// TIA Portal V16 export
// export: Created 2021-11-12T13:31:08.2127898Z, ExportSetting WithDefaults, DisplayName Totally Integrated Automation Portal, DisplayVersion V16 Update 3, DisplayName TIA Portal Version Control Interface, DisplayVersion V16 Update 2, DisplayName TIA Portal Openness, DisplayVersion V16 Update 3, DisplayName SINAMICS Startdrive Advanced, DisplayVersion V16 Update 5, DisplayName SINAMICS Startdrive G130, G150, S120, S150, SINAMICS MV, S210, DisplayVersion V16 Update 5, DisplayName SINAMICS Startdrive G110M, G120, G120C, G120D, G120P, G115D, DisplayVersion V16 Update 5, DisplayName STEP 7 Professional, DisplayVersion V16 Update 3, DisplayName STEP 7 Safety, DisplayVersion V16, DisplayName WinCC UA Professional, DisplayVersion V16 Update 3
FUNCTION_BLOCK "Main_Safety_RTG1"   // FB1, F_LAD
{ S7_Optimized_Access := 'TRUE' }
VERSION : 0.1
// stored: AutoNumber false, IsIECCheckEnabled false, UDAEnableTagReadback false
BEGIN

REGION Network 1: *************** Ingoing communication section start ***************
END_REGION

REGION Network 2: Communication: BSN1 / BSN2 -> CRS
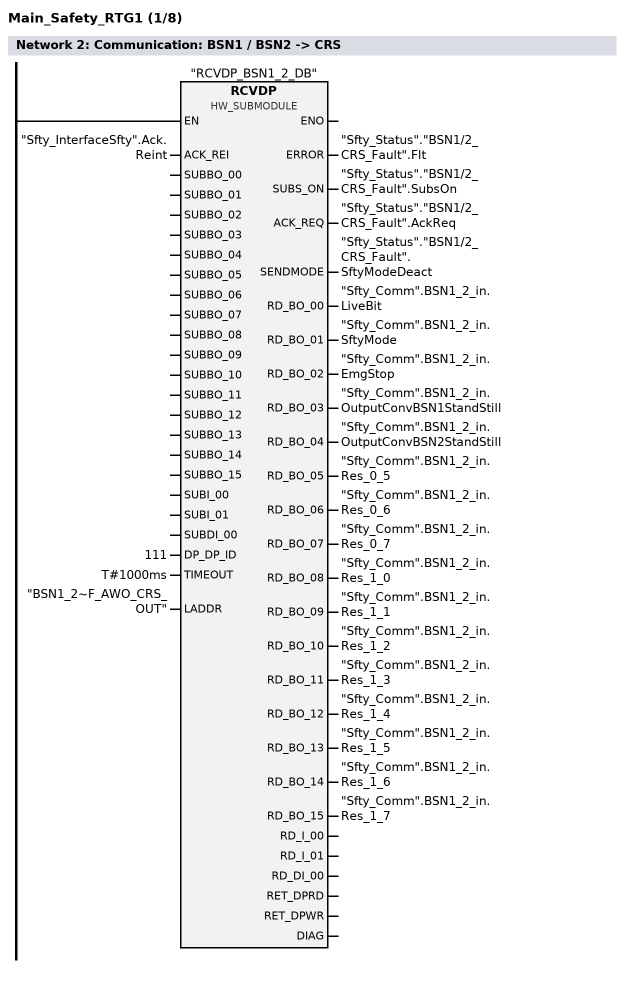
   RUNG wire#powerrail
      { S7_Templates := "laddr_type := HW_SUBMODULE" } "RCVDP_BSN1_2_DB".RCVDP(ACK_REI := "Sfty_InterfaceSfty".Ack.Reint, SUBBO_00 :=, SUBBO_01 :=, SUBBO_02 :=, SUBBO_03 :=, SUBBO_04 :=, SUBBO_05 :=, SUBBO_06 :=, SUBBO_07 :=, SUBBO_08 :=, SUBBO_09 :=, SUBBO_10 :=, SUBBO_11 :=, SUBBO_12 :=, SUBBO_13 :=, SUBBO_14 :=, SUBBO_15 :=, SUBI_00 :=, SUBI_01 :=, SUBDI_00 :=, DP_DP_ID := 111, TIMEOUT := T#1000ms, LADDR := "BSN1_2~F_AWO_CRS_OUT", ERROR => "Sfty_Status"."BSN1/2_CRS_Fault".Flt, SUBS_ON => "Sfty_Status"."BSN1/2_CRS_Fault".SubsOn, ACK_REQ => "Sfty_Status"."BSN1/2_CRS_Fault".AckReq, SENDMODE => "Sfty_Status"."BSN1/2_CRS_Fault".SftyModeDeact, RD_BO_00 => "Sfty_Comm".BSN1_2_in.LiveBit, RD_BO_01 => "Sfty_Comm".BSN1_2_in.SftyMode, RD_BO_02 => "Sfty_Comm".BSN1_2_in.EmgStop, RD_BO_03 => "Sfty_Comm".BSN1_2_in.OutputConvBSN1StandStill, RD_BO_04 => "Sfty_Comm".BSN1_2_in.OutputConvBSN2StandStill, RD_BO_05 => "Sfty_Comm".BSN1_2_in.Res_0_5, RD_BO_06 => "Sfty_Comm".BSN1_2_in.Res_0_6, RD_BO_07 => "Sfty_Comm".BSN1_2_in.Res_0_7, RD_BO_08 => "Sfty_Comm".BSN1_2_in.Res_1_0, RD_BO_09 => "Sfty_Comm".BSN1_2_in.Res_1_1, RD_BO_10 => "Sfty_Comm".BSN1_2_in.Res_1_2, RD_BO_11 => "Sfty_Comm".BSN1_2_in.Res_1_3, RD_BO_12 => "Sfty_Comm".BSN1_2_in.Res_1_4, RD_BO_13 => "Sfty_Comm".BSN1_2_in.Res_1_5, RD_BO_14 => "Sfty_Comm".BSN1_2_in.Res_1_6, RD_BO_15 => "Sfty_Comm".BSN1_2_in.Res_1_7, RD_I_00 =>, RD_I_01 =>, RD_DI_00 =>, RET_DPRD =>, RET_DPWR =>, DIAG =>)
   END_RUNG
   // the same network as SCL:
   "RCVDP_BSN1_2_DB"(ACK_REI := "Sfty_InterfaceSfty".Ack.Reint,   // RCVDP
                     DP_DP_ID := 111,
                     TIMEOUT := T#1000ms,
                     LADDR := "BSN1_2~F_AWO_CRS_OUT",
                     ERROR => "Sfty_Status"."BSN1/2_CRS_Fault".Flt,
                     SUBS_ON => "Sfty_Status"."BSN1/2_CRS_Fault".SubsOn,
                     ACK_REQ => "Sfty_Status"."BSN1/2_CRS_Fault".AckReq,
                     SENDMODE => "Sfty_Status"."BSN1/2_CRS_Fault".SftyModeDeact,
                     RD_BO_00 => "Sfty_Comm".BSN1_2_in.LiveBit,
                     RD_BO_01 => "Sfty_Comm".BSN1_2_in.SftyMode,
                     RD_BO_02 => "Sfty_Comm".BSN1_2_in.EmgStop,
                     RD_BO_03 => "Sfty_Comm".BSN1_2_in.OutputConvBSN1StandStill,
                     RD_BO_04 => "Sfty_Comm".BSN1_2_in.OutputConvBSN2StandStill,
                     RD_BO_05 => "Sfty_Comm".BSN1_2_in.Res_0_5,
                     RD_BO_06 => "Sfty_Comm".BSN1_2_in.Res_0_6,
                     RD_BO_07 => "Sfty_Comm".BSN1_2_in.Res_0_7,
                     RD_BO_08 => "Sfty_Comm".BSN1_2_in.Res_1_0,
                     RD_BO_09 => "Sfty_Comm".BSN1_2_in.Res_1_1,
                     RD_BO_10 => "Sfty_Comm".BSN1_2_in.Res_1_2,
                     RD_BO_11 => "Sfty_Comm".BSN1_2_in.Res_1_3,
                     RD_BO_12 => "Sfty_Comm".BSN1_2_in.Res_1_4,
                     RD_BO_13 => "Sfty_Comm".BSN1_2_in.Res_1_5,
                     RD_BO_14 => "Sfty_Comm".BSN1_2_in.Res_1_6,
                     RD_BO_15 => "Sfty_Comm".BSN1_2_in.Res_1_7);
END_REGION

REGION Network 3: Communication: SCH1 -> CRS
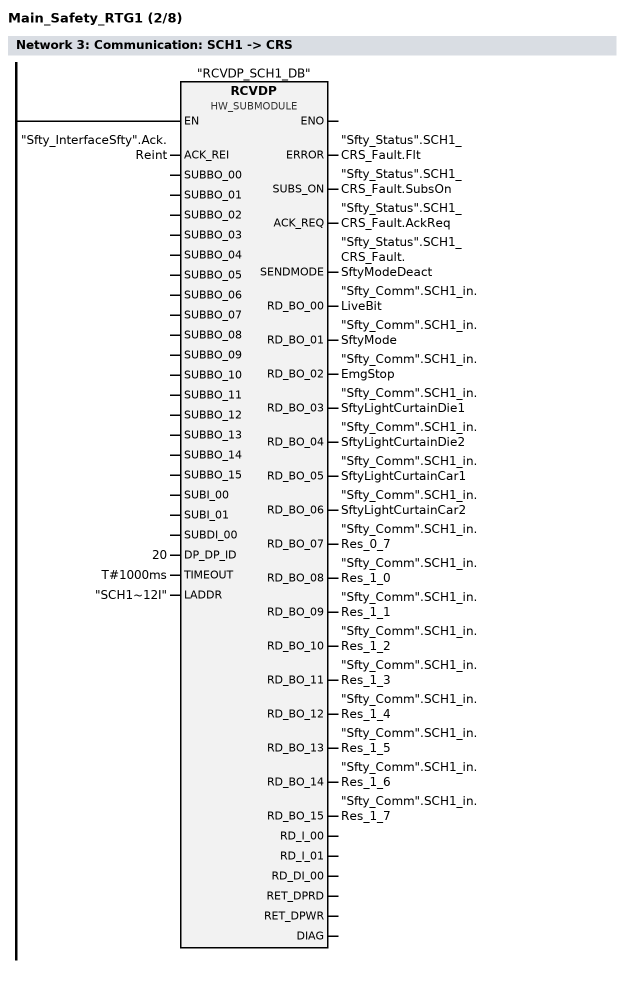
   RUNG wire#powerrail
      { S7_Templates := "laddr_type := HW_SUBMODULE" } "RCVDP_SCH1_DB".RCVDP(ACK_REI := "Sfty_InterfaceSfty".Ack.Reint, SUBBO_00 :=, SUBBO_01 :=, SUBBO_02 :=, SUBBO_03 :=, SUBBO_04 :=, SUBBO_05 :=, SUBBO_06 :=, SUBBO_07 :=, SUBBO_08 :=, SUBBO_09 :=, SUBBO_10 :=, SUBBO_11 :=, SUBBO_12 :=, SUBBO_13 :=, SUBBO_14 :=, SUBBO_15 :=, SUBI_00 :=, SUBI_01 :=, SUBDI_00 :=, DP_DP_ID := 20, TIMEOUT := T#1000ms, LADDR := "SCH1~12I", ERROR => "Sfty_Status".SCH1_CRS_Fault.Flt, SUBS_ON => "Sfty_Status".SCH1_CRS_Fault.SubsOn, ACK_REQ => "Sfty_Status".SCH1_CRS_Fault.AckReq, SENDMODE => "Sfty_Status".SCH1_CRS_Fault.SftyModeDeact, RD_BO_00 => "Sfty_Comm".SCH1_in.LiveBit, RD_BO_01 => "Sfty_Comm".SCH1_in.SftyMode, RD_BO_02 => "Sfty_Comm".SCH1_in.EmgStop, RD_BO_03 => "Sfty_Comm".SCH1_in.SftyLightCurtainDie1, RD_BO_04 => "Sfty_Comm".SCH1_in.SftyLightCurtainDie2, RD_BO_05 => "Sfty_Comm".SCH1_in.SftyLightCurtainCar1, RD_BO_06 => "Sfty_Comm".SCH1_in.SftyLightCurtainCar2, RD_BO_07 => "Sfty_Comm".SCH1_in.Res_0_7, RD_BO_08 => "Sfty_Comm".SCH1_in.Res_1_0, RD_BO_09 => "Sfty_Comm".SCH1_in.Res_1_1, RD_BO_10 => "Sfty_Comm".SCH1_in.Res_1_2, RD_BO_11 => "Sfty_Comm".SCH1_in.Res_1_3, RD_BO_12 => "Sfty_Comm".SCH1_in.Res_1_4, RD_BO_13 => "Sfty_Comm".SCH1_in.Res_1_5, RD_BO_14 => "Sfty_Comm".SCH1_in.Res_1_6, RD_BO_15 => "Sfty_Comm".SCH1_in.Res_1_7, RD_I_00 =>, RD_I_01 =>, RD_DI_00 =>, RET_DPRD =>, RET_DPWR =>, DIAG =>)
   END_RUNG
   // the same network as SCL:
   "RCVDP_SCH1_DB"(ACK_REI := "Sfty_InterfaceSfty".Ack.Reint,   // RCVDP
                   DP_DP_ID := 20,
                   TIMEOUT := T#1000ms,
                   LADDR := "SCH1~12I",
                   ERROR => "Sfty_Status".SCH1_CRS_Fault.Flt,
                   SUBS_ON => "Sfty_Status".SCH1_CRS_Fault.SubsOn,
                   ACK_REQ => "Sfty_Status".SCH1_CRS_Fault.AckReq,
                   SENDMODE => "Sfty_Status".SCH1_CRS_Fault.SftyModeDeact,
                   RD_BO_00 => "Sfty_Comm".SCH1_in.LiveBit,
                   RD_BO_01 => "Sfty_Comm".SCH1_in.SftyMode,
                   RD_BO_02 => "Sfty_Comm".SCH1_in.EmgStop,
                   RD_BO_03 => "Sfty_Comm".SCH1_in.SftyLightCurtainDie1,
                   RD_BO_04 => "Sfty_Comm".SCH1_in.SftyLightCurtainDie2,
                   RD_BO_05 => "Sfty_Comm".SCH1_in.SftyLightCurtainCar1,
                   RD_BO_06 => "Sfty_Comm".SCH1_in.SftyLightCurtainCar2,
                   RD_BO_07 => "Sfty_Comm".SCH1_in.Res_0_7,
                   RD_BO_08 => "Sfty_Comm".SCH1_in.Res_1_0,
                   RD_BO_09 => "Sfty_Comm".SCH1_in.Res_1_1,
                   RD_BO_10 => "Sfty_Comm".SCH1_in.Res_1_2,
                   RD_BO_11 => "Sfty_Comm".SCH1_in.Res_1_3,
                   RD_BO_12 => "Sfty_Comm".SCH1_in.Res_1_4,
                   RD_BO_13 => "Sfty_Comm".SCH1_in.Res_1_5,
                   RD_BO_14 => "Sfty_Comm".SCH1_in.Res_1_6,
                   RD_BO_15 => "Sfty_Comm".SCH1_in.Res_1_7);
END_REGION

REGION Network 4: Communication: BSN3 -> CRS
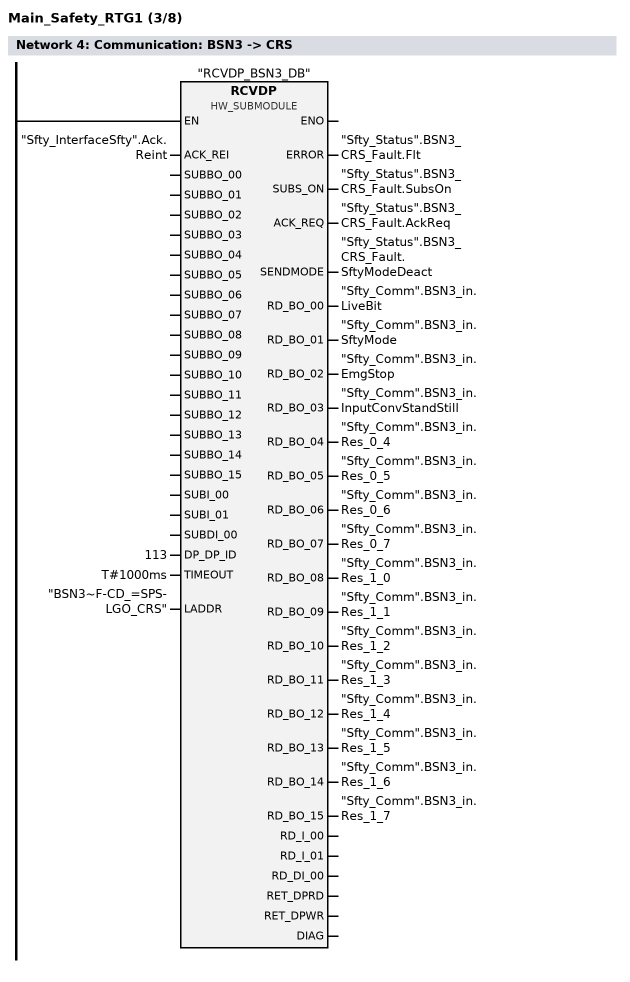
   RUNG wire#powerrail
      { S7_Templates := "laddr_type := HW_SUBMODULE" } "RCVDP_BSN3_DB".RCVDP(ACK_REI := "Sfty_InterfaceSfty".Ack.Reint, SUBBO_00 :=, SUBBO_01 :=, SUBBO_02 :=, SUBBO_03 :=, SUBBO_04 :=, SUBBO_05 :=, SUBBO_06 :=, SUBBO_07 :=, SUBBO_08 :=, SUBBO_09 :=, SUBBO_10 :=, SUBBO_11 :=, SUBBO_12 :=, SUBBO_13 :=, SUBBO_14 :=, SUBBO_15 :=, SUBI_00 :=, SUBI_01 :=, SUBDI_00 :=, DP_DP_ID := 113, TIMEOUT := T#1000ms, LADDR := "BSN3~F-CD_=SPS-LGO_CRS", ERROR => "Sfty_Status".BSN3_CRS_Fault.Flt, SUBS_ON => "Sfty_Status".BSN3_CRS_Fault.SubsOn, ACK_REQ => "Sfty_Status".BSN3_CRS_Fault.AckReq, SENDMODE => "Sfty_Status".BSN3_CRS_Fault.SftyModeDeact, RD_BO_00 => "Sfty_Comm".BSN3_in.LiveBit, RD_BO_01 => "Sfty_Comm".BSN3_in.SftyMode, RD_BO_02 => "Sfty_Comm".BSN3_in.EmgStop, RD_BO_03 => "Sfty_Comm".BSN3_in.InputConvStandStill, RD_BO_04 => "Sfty_Comm".BSN3_in.Res_0_4, RD_BO_05 => "Sfty_Comm".BSN3_in.Res_0_5, RD_BO_06 => "Sfty_Comm".BSN3_in.Res_0_6, RD_BO_07 => "Sfty_Comm".BSN3_in.Res_0_7, RD_BO_08 => "Sfty_Comm".BSN3_in.Res_1_0, RD_BO_09 => "Sfty_Comm".BSN3_in.Res_1_1, RD_BO_10 => "Sfty_Comm".BSN3_in.Res_1_2, RD_BO_11 => "Sfty_Comm".BSN3_in.Res_1_3, RD_BO_12 => "Sfty_Comm".BSN3_in.Res_1_4, RD_BO_13 => "Sfty_Comm".BSN3_in.Res_1_5, RD_BO_14 => "Sfty_Comm".BSN3_in.Res_1_6, RD_BO_15 => "Sfty_Comm".BSN3_in.Res_1_7, RD_I_00 =>, RD_I_01 =>, RD_DI_00 =>, RET_DPRD =>, RET_DPWR =>, DIAG =>)
   END_RUNG
   // the same network as SCL:
   "RCVDP_BSN3_DB"(ACK_REI := "Sfty_InterfaceSfty".Ack.Reint,   // RCVDP
                   DP_DP_ID := 113,
                   TIMEOUT := T#1000ms,
                   LADDR := "BSN3~F-CD_=SPS-LGO_CRS",
                   ERROR => "Sfty_Status".BSN3_CRS_Fault.Flt,
                   SUBS_ON => "Sfty_Status".BSN3_CRS_Fault.SubsOn,
                   ACK_REQ => "Sfty_Status".BSN3_CRS_Fault.AckReq,
                   SENDMODE => "Sfty_Status".BSN3_CRS_Fault.SftyModeDeact,
                   RD_BO_00 => "Sfty_Comm".BSN3_in.LiveBit,
                   RD_BO_01 => "Sfty_Comm".BSN3_in.SftyMode,
                   RD_BO_02 => "Sfty_Comm".BSN3_in.EmgStop,
                   RD_BO_03 => "Sfty_Comm".BSN3_in.InputConvStandStill,
                   RD_BO_04 => "Sfty_Comm".BSN3_in.Res_0_4,
                   RD_BO_05 => "Sfty_Comm".BSN3_in.Res_0_5,
                   RD_BO_06 => "Sfty_Comm".BSN3_in.Res_0_6,
                   RD_BO_07 => "Sfty_Comm".BSN3_in.Res_0_7,
                   RD_BO_08 => "Sfty_Comm".BSN3_in.Res_1_0,
                   RD_BO_09 => "Sfty_Comm".BSN3_in.Res_1_1,
                   RD_BO_10 => "Sfty_Comm".BSN3_in.Res_1_2,
                   RD_BO_11 => "Sfty_Comm".BSN3_in.Res_1_3,
                   RD_BO_12 => "Sfty_Comm".BSN3_in.Res_1_4,
                   RD_BO_13 => "Sfty_Comm".BSN3_in.Res_1_5,
                   RD_BO_14 => "Sfty_Comm".BSN3_in.Res_1_6,
                   RD_BO_15 => "Sfty_Comm".BSN3_in.Res_1_7);
END_REGION

REGION Network 5: Communication: BSN4 / BSN5 -> CRS
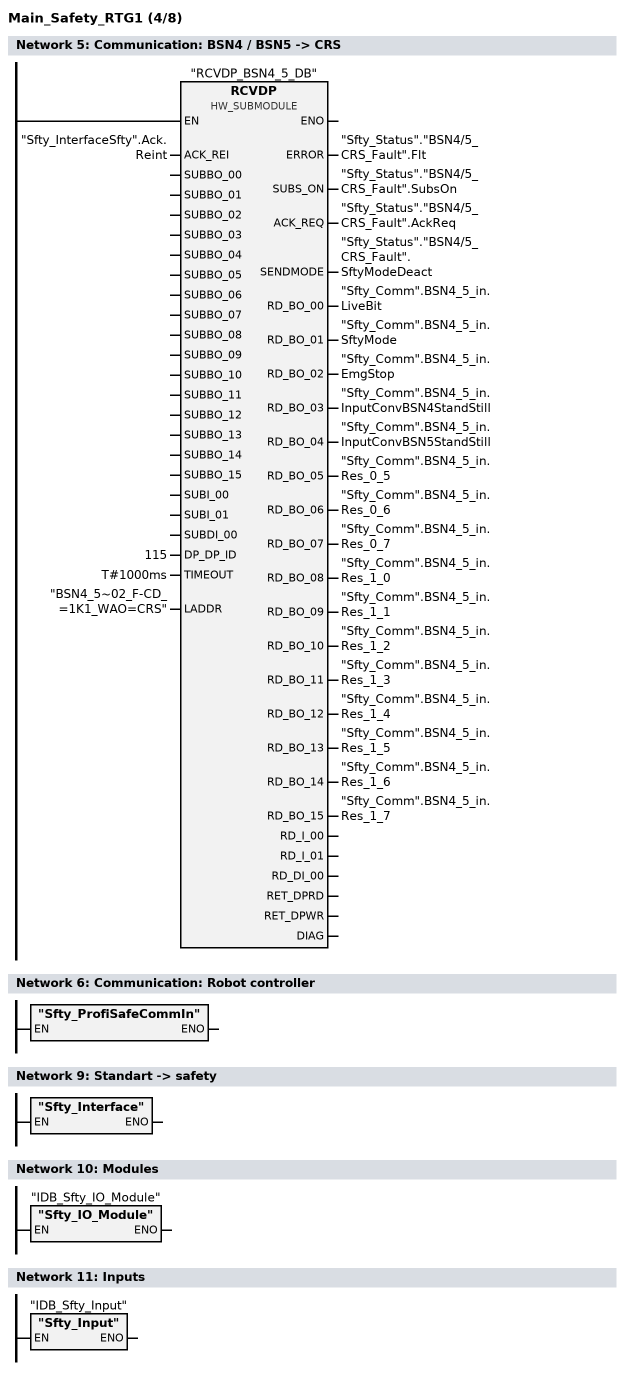
   RUNG wire#powerrail
      { S7_Templates := "laddr_type := HW_SUBMODULE" } "RCVDP_BSN4_5_DB".RCVDP(ACK_REI := "Sfty_InterfaceSfty".Ack.Reint, SUBBO_00 :=, SUBBO_01 :=, SUBBO_02 :=, SUBBO_03 :=, SUBBO_04 :=, SUBBO_05 :=, SUBBO_06 :=, SUBBO_07 :=, SUBBO_08 :=, SUBBO_09 :=, SUBBO_10 :=, SUBBO_11 :=, SUBBO_12 :=, SUBBO_13 :=, SUBBO_14 :=, SUBBO_15 :=, SUBI_00 :=, SUBI_01 :=, SUBDI_00 :=, DP_DP_ID := 115, TIMEOUT := T#1000ms, LADDR := "BSN4_5~02_F-CD_=1K1_WAO=CRS", ERROR => "Sfty_Status"."BSN4/5_CRS_Fault".Flt, SUBS_ON => "Sfty_Status"."BSN4/5_CRS_Fault".SubsOn, ACK_REQ => "Sfty_Status"."BSN4/5_CRS_Fault".AckReq, SENDMODE => "Sfty_Status"."BSN4/5_CRS_Fault".SftyModeDeact, RD_BO_00 => "Sfty_Comm".BSN4_5_in.LiveBit, RD_BO_01 => "Sfty_Comm".BSN4_5_in.SftyMode, RD_BO_02 => "Sfty_Comm".BSN4_5_in.EmgStop, RD_BO_03 => "Sfty_Comm".BSN4_5_in.InputConvBSN4StandStill, RD_BO_04 => "Sfty_Comm".BSN4_5_in.InputConvBSN5StandStill, RD_BO_05 => "Sfty_Comm".BSN4_5_in.Res_0_5, RD_BO_06 => "Sfty_Comm".BSN4_5_in.Res_0_6, RD_BO_07 => "Sfty_Comm".BSN4_5_in.Res_0_7, RD_BO_08 => "Sfty_Comm".BSN4_5_in.Res_1_0, RD_BO_09 => "Sfty_Comm".BSN4_5_in.Res_1_1, RD_BO_10 => "Sfty_Comm".BSN4_5_in.Res_1_2, RD_BO_11 => "Sfty_Comm".BSN4_5_in.Res_1_3, RD_BO_12 => "Sfty_Comm".BSN4_5_in.Res_1_4, RD_BO_13 => "Sfty_Comm".BSN4_5_in.Res_1_5, RD_BO_14 => "Sfty_Comm".BSN4_5_in.Res_1_6, RD_BO_15 => "Sfty_Comm".BSN4_5_in.Res_1_7, RD_I_00 =>, RD_I_01 =>, RD_DI_00 =>, RET_DPRD =>, RET_DPWR =>, DIAG =>)
   END_RUNG
   // the same network as SCL:
   "RCVDP_BSN4_5_DB"(ACK_REI := "Sfty_InterfaceSfty".Ack.Reint,   // RCVDP
                     DP_DP_ID := 115,
                     TIMEOUT := T#1000ms,
                     LADDR := "BSN4_5~02_F-CD_=1K1_WAO=CRS",
                     ERROR => "Sfty_Status"."BSN4/5_CRS_Fault".Flt,
                     SUBS_ON => "Sfty_Status"."BSN4/5_CRS_Fault".SubsOn,
                     ACK_REQ => "Sfty_Status"."BSN4/5_CRS_Fault".AckReq,
                     SENDMODE => "Sfty_Status"."BSN4/5_CRS_Fault".SftyModeDeact,
                     RD_BO_00 => "Sfty_Comm".BSN4_5_in.LiveBit,
                     RD_BO_01 => "Sfty_Comm".BSN4_5_in.SftyMode,
                     RD_BO_02 => "Sfty_Comm".BSN4_5_in.EmgStop,
                     RD_BO_03 => "Sfty_Comm".BSN4_5_in.InputConvBSN4StandStill,
                     RD_BO_04 => "Sfty_Comm".BSN4_5_in.InputConvBSN5StandStill,
                     RD_BO_05 => "Sfty_Comm".BSN4_5_in.Res_0_5,
                     RD_BO_06 => "Sfty_Comm".BSN4_5_in.Res_0_6,
                     RD_BO_07 => "Sfty_Comm".BSN4_5_in.Res_0_7,
                     RD_BO_08 => "Sfty_Comm".BSN4_5_in.Res_1_0,
                     RD_BO_09 => "Sfty_Comm".BSN4_5_in.Res_1_1,
                     RD_BO_10 => "Sfty_Comm".BSN4_5_in.Res_1_2,
                     RD_BO_11 => "Sfty_Comm".BSN4_5_in.Res_1_3,
                     RD_BO_12 => "Sfty_Comm".BSN4_5_in.Res_1_4,
                     RD_BO_13 => "Sfty_Comm".BSN4_5_in.Res_1_5,
                     RD_BO_14 => "Sfty_Comm".BSN4_5_in.Res_1_6,
                     RD_BO_15 => "Sfty_Comm".BSN4_5_in.Res_1_7);
END_REGION

REGION Network 6: Communication: Robot controller
   RUNG wire#powerrail
      "Sfty_ProfiSafeCommIn"()
   END_RUNG
   // the same network as SCL:
   "Sfty_ProfiSafeCommIn"();
END_REGION

REGION Network 7: *************** Ingoing communication section end ***************
END_REGION

REGION Network 8: *************** Interface ***************
END_REGION

REGION Network 9: Standart -> safety
   RUNG wire#powerrail
      "Sfty_Interface"()
   END_RUNG
   // the same network as SCL:
   "Sfty_Interface"();
END_REGION

REGION Network 10: Modules
   RUNG wire#powerrail
      "IDB_Sfty_IO_Module"()
   END_RUNG
   // the same network as SCL:
   "IDB_Sfty_IO_Module"();   // "Sfty_IO_Module"
END_REGION

REGION Network 11: Inputs
   RUNG wire#powerrail
      "IDB_Sfty_Input"()
   END_RUNG
   // the same network as SCL:
   "IDB_Sfty_Input"();   // "Sfty_Input"
END_REGION

REGION Network 12: Outputs
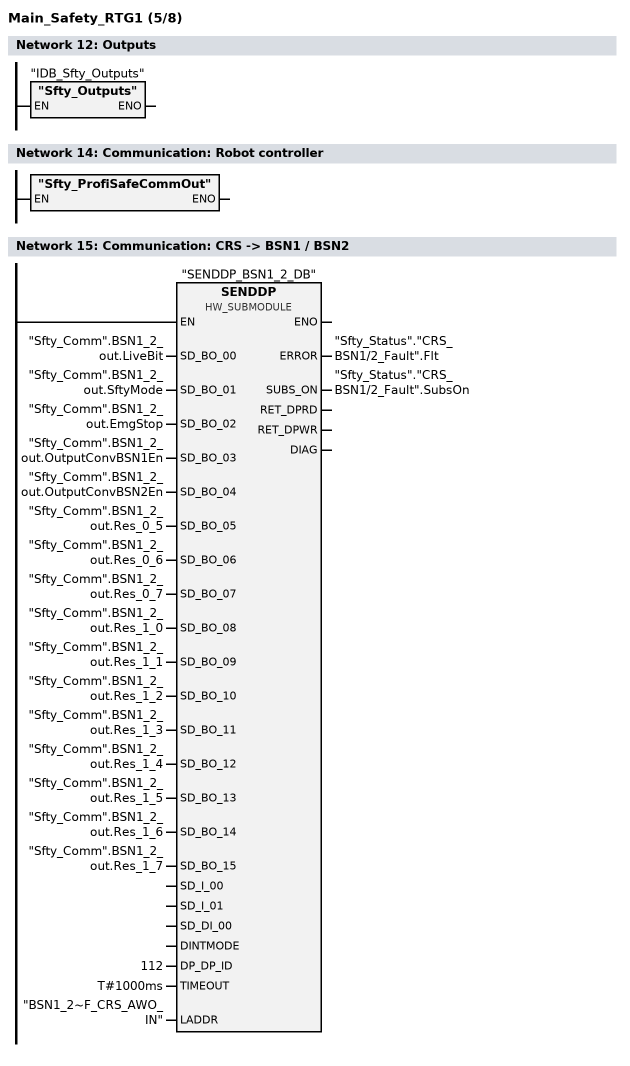
   RUNG wire#powerrail
      "IDB_Sfty_Outputs"()
   END_RUNG
   // the same network as SCL:
   "IDB_Sfty_Outputs"();   // "Sfty_Outputs"
END_REGION

REGION Network 13: *************** Outgoing communication section start ***************
END_REGION

REGION Network 14: Communication: Robot controller
   RUNG wire#powerrail
      "Sfty_ProfiSafeCommOut"()
   END_RUNG
   // the same network as SCL:
   "Sfty_ProfiSafeCommOut"();
END_REGION

REGION Network 15: Communication: CRS -> BSN1 / BSN2
   RUNG wire#powerrail
      { S7_Templates := "laddr_type := HW_SUBMODULE" } "SENDDP_BSN1_2_DB".SENDDP(SD_BO_00 := "Sfty_Comm".BSN1_2_out.LiveBit, SD_BO_01 := "Sfty_Comm".BSN1_2_out.SftyMode, SD_BO_02 := "Sfty_Comm".BSN1_2_out.EmgStop, SD_BO_03 := "Sfty_Comm".BSN1_2_out.OutputConvBSN1En, SD_BO_04 := "Sfty_Comm".BSN1_2_out.OutputConvBSN2En, SD_BO_05 := "Sfty_Comm".BSN1_2_out.Res_0_5, SD_BO_06 := "Sfty_Comm".BSN1_2_out.Res_0_6, SD_BO_07 := "Sfty_Comm".BSN1_2_out.Res_0_7, SD_BO_08 := "Sfty_Comm".BSN1_2_out.Res_1_0, SD_BO_09 := "Sfty_Comm".BSN1_2_out.Res_1_1, SD_BO_10 := "Sfty_Comm".BSN1_2_out.Res_1_2, SD_BO_11 := "Sfty_Comm".BSN1_2_out.Res_1_3, SD_BO_12 := "Sfty_Comm".BSN1_2_out.Res_1_4, SD_BO_13 := "Sfty_Comm".BSN1_2_out.Res_1_5, SD_BO_14 := "Sfty_Comm".BSN1_2_out.Res_1_6, SD_BO_15 := "Sfty_Comm".BSN1_2_out.Res_1_7, SD_I_00 :=, SD_I_01 :=, SD_DI_00 :=, DINTMODE :=, DP_DP_ID := 112, TIMEOUT := T#1000ms, LADDR := "BSN1_2~F_CRS_AWO_IN", ERROR => "Sfty_Status"."CRS_BSN1/2_Fault".Flt, SUBS_ON => "Sfty_Status"."CRS_BSN1/2_Fault".SubsOn, RET_DPRD =>, RET_DPWR =>, DIAG =>)
   END_RUNG
   // the same network as SCL:
   "SENDDP_BSN1_2_DB"(SD_BO_00 := "Sfty_Comm".BSN1_2_out.LiveBit,   // SENDDP
                      SD_BO_01 := "Sfty_Comm".BSN1_2_out.SftyMode,
                      SD_BO_02 := "Sfty_Comm".BSN1_2_out.EmgStop,
                      SD_BO_03 := "Sfty_Comm".BSN1_2_out.OutputConvBSN1En,
                      SD_BO_04 := "Sfty_Comm".BSN1_2_out.OutputConvBSN2En,
                      SD_BO_05 := "Sfty_Comm".BSN1_2_out.Res_0_5,
                      SD_BO_06 := "Sfty_Comm".BSN1_2_out.Res_0_6,
                      SD_BO_07 := "Sfty_Comm".BSN1_2_out.Res_0_7,
                      SD_BO_08 := "Sfty_Comm".BSN1_2_out.Res_1_0,
                      SD_BO_09 := "Sfty_Comm".BSN1_2_out.Res_1_1,
                      SD_BO_10 := "Sfty_Comm".BSN1_2_out.Res_1_2,
                      SD_BO_11 := "Sfty_Comm".BSN1_2_out.Res_1_3,
                      SD_BO_12 := "Sfty_Comm".BSN1_2_out.Res_1_4,
                      SD_BO_13 := "Sfty_Comm".BSN1_2_out.Res_1_5,
                      SD_BO_14 := "Sfty_Comm".BSN1_2_out.Res_1_6,
                      SD_BO_15 := "Sfty_Comm".BSN1_2_out.Res_1_7,
                      DP_DP_ID := 112,
                      TIMEOUT := T#1000ms,
                      LADDR := "BSN1_2~F_CRS_AWO_IN",
                      ERROR => "Sfty_Status"."CRS_BSN1/2_Fault".Flt,
                      SUBS_ON => "Sfty_Status"."CRS_BSN1/2_Fault".SubsOn);
END_REGION

REGION Network 16: Communication: CRS -> SCH1
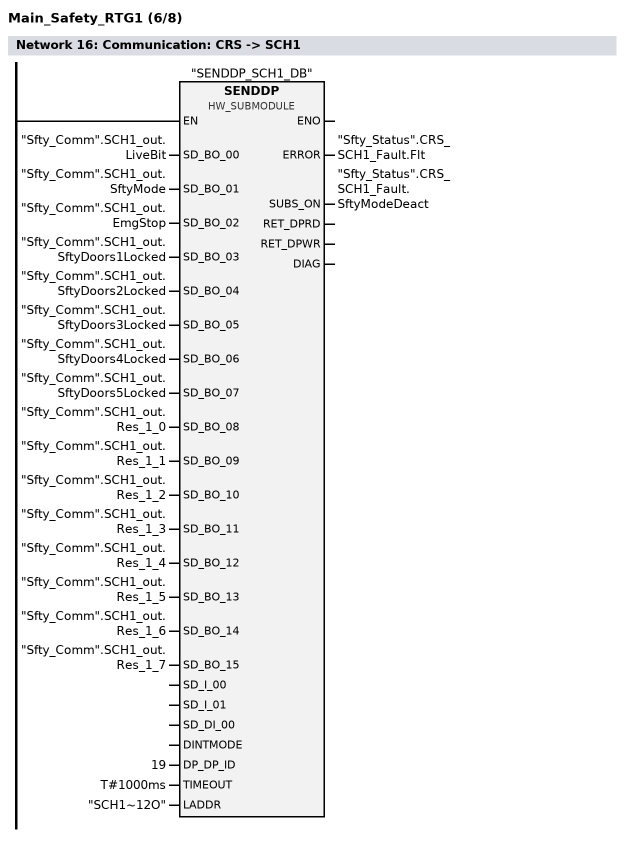
   RUNG wire#powerrail
      { S7_Templates := "laddr_type := HW_SUBMODULE" } "SENDDP_SCH1_DB".SENDDP(SD_BO_00 := "Sfty_Comm".SCH1_out.LiveBit, SD_BO_01 := "Sfty_Comm".SCH1_out.SftyMode, SD_BO_02 := "Sfty_Comm".SCH1_out.EmgStop, SD_BO_03 := "Sfty_Comm".SCH1_out.SftyDoors1Locked, SD_BO_04 := "Sfty_Comm".SCH1_out.SftyDoors2Locked, SD_BO_05 := "Sfty_Comm".SCH1_out.SftyDoors3Locked, SD_BO_06 := "Sfty_Comm".SCH1_out.SftyDoors4Locked, SD_BO_07 := "Sfty_Comm".SCH1_out.SftyDoors5Locked, SD_BO_08 := "Sfty_Comm".SCH1_out.Res_1_0, SD_BO_09 := "Sfty_Comm".SCH1_out.Res_1_1, SD_BO_10 := "Sfty_Comm".SCH1_out.Res_1_2, SD_BO_11 := "Sfty_Comm".SCH1_out.Res_1_3, SD_BO_12 := "Sfty_Comm".SCH1_out.Res_1_4, SD_BO_13 := "Sfty_Comm".SCH1_out.Res_1_5, SD_BO_14 := "Sfty_Comm".SCH1_out.Res_1_6, SD_BO_15 := "Sfty_Comm".SCH1_out.Res_1_7, SD_I_00 :=, SD_I_01 :=, SD_DI_00 :=, DINTMODE :=, DP_DP_ID := 19, TIMEOUT := T#1000ms, LADDR := "SCH1~12O", ERROR => "Sfty_Status".CRS_SCH1_Fault.Flt, SUBS_ON => "Sfty_Status".CRS_SCH1_Fault.SftyModeDeact, RET_DPRD =>, RET_DPWR =>, DIAG =>)
   END_RUNG
   // the same network as SCL:
   "SENDDP_SCH1_DB"(SD_BO_00 := "Sfty_Comm".SCH1_out.LiveBit,   // SENDDP
                    SD_BO_01 := "Sfty_Comm".SCH1_out.SftyMode,
                    SD_BO_02 := "Sfty_Comm".SCH1_out.EmgStop,
                    SD_BO_03 := "Sfty_Comm".SCH1_out.SftyDoors1Locked,
                    SD_BO_04 := "Sfty_Comm".SCH1_out.SftyDoors2Locked,
                    SD_BO_05 := "Sfty_Comm".SCH1_out.SftyDoors3Locked,
                    SD_BO_06 := "Sfty_Comm".SCH1_out.SftyDoors4Locked,
                    SD_BO_07 := "Sfty_Comm".SCH1_out.SftyDoors5Locked,
                    SD_BO_08 := "Sfty_Comm".SCH1_out.Res_1_0,
                    SD_BO_09 := "Sfty_Comm".SCH1_out.Res_1_1,
                    SD_BO_10 := "Sfty_Comm".SCH1_out.Res_1_2,
                    SD_BO_11 := "Sfty_Comm".SCH1_out.Res_1_3,
                    SD_BO_12 := "Sfty_Comm".SCH1_out.Res_1_4,
                    SD_BO_13 := "Sfty_Comm".SCH1_out.Res_1_5,
                    SD_BO_14 := "Sfty_Comm".SCH1_out.Res_1_6,
                    SD_BO_15 := "Sfty_Comm".SCH1_out.Res_1_7,
                    DP_DP_ID := 19,
                    TIMEOUT := T#1000ms,
                    LADDR := "SCH1~12O",
                    ERROR => "Sfty_Status".CRS_SCH1_Fault.Flt,
                    SUBS_ON => "Sfty_Status".CRS_SCH1_Fault.SftyModeDeact);
END_REGION

REGION Network 17: Communication: CRS -> BSN3
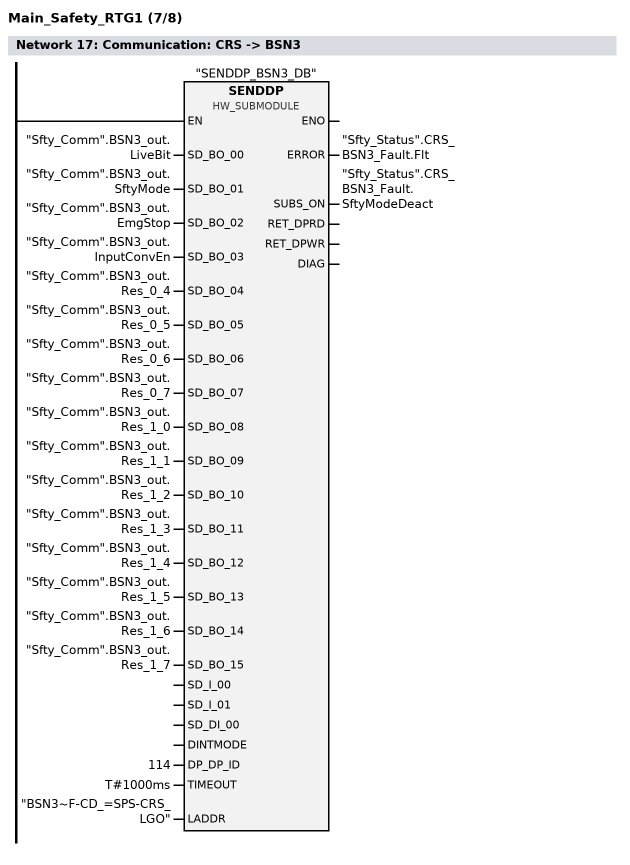
   RUNG wire#powerrail
      { S7_Templates := "laddr_type := HW_SUBMODULE" } "SENDDP_BSN3_DB".SENDDP(SD_BO_00 := "Sfty_Comm".BSN3_out.LiveBit, SD_BO_01 := "Sfty_Comm".BSN3_out.SftyMode, SD_BO_02 := "Sfty_Comm".BSN3_out.EmgStop, SD_BO_03 := "Sfty_Comm".BSN3_out.InputConvEn, SD_BO_04 := "Sfty_Comm".BSN3_out.Res_0_4, SD_BO_05 := "Sfty_Comm".BSN3_out.Res_0_5, SD_BO_06 := "Sfty_Comm".BSN3_out.Res_0_6, SD_BO_07 := "Sfty_Comm".BSN3_out.Res_0_7, SD_BO_08 := "Sfty_Comm".BSN3_out.Res_1_0, SD_BO_09 := "Sfty_Comm".BSN3_out.Res_1_1, SD_BO_10 := "Sfty_Comm".BSN3_out.Res_1_2, SD_BO_11 := "Sfty_Comm".BSN3_out.Res_1_3, SD_BO_12 := "Sfty_Comm".BSN3_out.Res_1_4, SD_BO_13 := "Sfty_Comm".BSN3_out.Res_1_5, SD_BO_14 := "Sfty_Comm".BSN3_out.Res_1_6, SD_BO_15 := "Sfty_Comm".BSN3_out.Res_1_7, SD_I_00 :=, SD_I_01 :=, SD_DI_00 :=, DINTMODE :=, DP_DP_ID := 114, TIMEOUT := T#1000ms, LADDR := "BSN3~F-CD_=SPS-CRS_LGO", ERROR => "Sfty_Status".CRS_BSN3_Fault.Flt, SUBS_ON => "Sfty_Status".CRS_BSN3_Fault.SftyModeDeact, RET_DPRD =>, RET_DPWR =>, DIAG =>)
   END_RUNG
   // the same network as SCL:
   "SENDDP_BSN3_DB"(SD_BO_00 := "Sfty_Comm".BSN3_out.LiveBit,   // SENDDP
                    SD_BO_01 := "Sfty_Comm".BSN3_out.SftyMode,
                    SD_BO_02 := "Sfty_Comm".BSN3_out.EmgStop,
                    SD_BO_03 := "Sfty_Comm".BSN3_out.InputConvEn,
                    SD_BO_04 := "Sfty_Comm".BSN3_out.Res_0_4,
                    SD_BO_05 := "Sfty_Comm".BSN3_out.Res_0_5,
                    SD_BO_06 := "Sfty_Comm".BSN3_out.Res_0_6,
                    SD_BO_07 := "Sfty_Comm".BSN3_out.Res_0_7,
                    SD_BO_08 := "Sfty_Comm".BSN3_out.Res_1_0,
                    SD_BO_09 := "Sfty_Comm".BSN3_out.Res_1_1,
                    SD_BO_10 := "Sfty_Comm".BSN3_out.Res_1_2,
                    SD_BO_11 := "Sfty_Comm".BSN3_out.Res_1_3,
                    SD_BO_12 := "Sfty_Comm".BSN3_out.Res_1_4,
                    SD_BO_13 := "Sfty_Comm".BSN3_out.Res_1_5,
                    SD_BO_14 := "Sfty_Comm".BSN3_out.Res_1_6,
                    SD_BO_15 := "Sfty_Comm".BSN3_out.Res_1_7,
                    DP_DP_ID := 114,
                    TIMEOUT := T#1000ms,
                    LADDR := "BSN3~F-CD_=SPS-CRS_LGO",
                    ERROR => "Sfty_Status".CRS_BSN3_Fault.Flt,
                    SUBS_ON => "Sfty_Status".CRS_BSN3_Fault.SftyModeDeact);
END_REGION

REGION Network 18: Communication: CRS -> BSN4 / BSN5
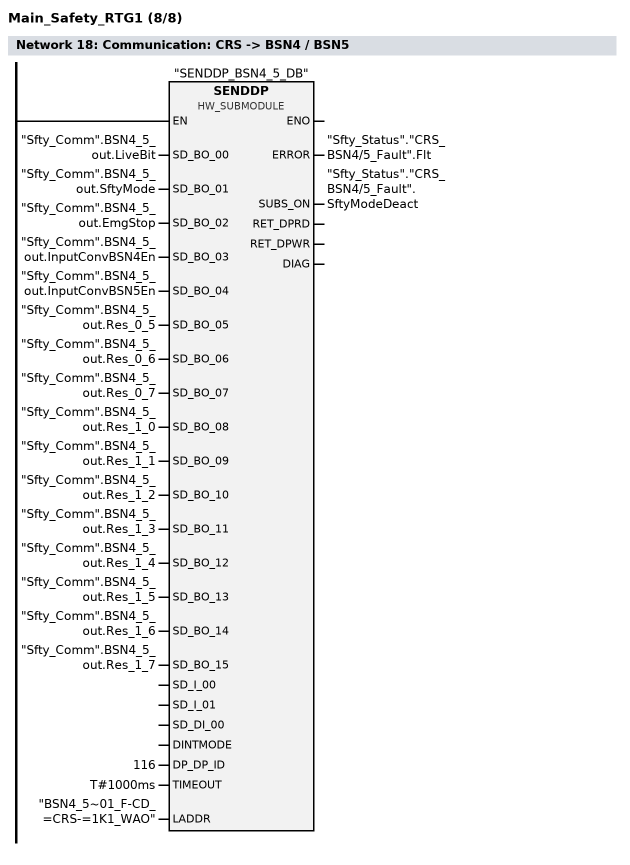
   RUNG wire#powerrail
      { S7_Templates := "laddr_type := HW_SUBMODULE" } "SENDDP_BSN4_5_DB".SENDDP(SD_BO_00 := "Sfty_Comm".BSN4_5_out.LiveBit, SD_BO_01 := "Sfty_Comm".BSN4_5_out.SftyMode, SD_BO_02 := "Sfty_Comm".BSN4_5_out.EmgStop, SD_BO_03 := "Sfty_Comm".BSN4_5_out.InputConvBSN4En, SD_BO_04 := "Sfty_Comm".BSN4_5_out.InputConvBSN5En, SD_BO_05 := "Sfty_Comm".BSN4_5_out.Res_0_5, SD_BO_06 := "Sfty_Comm".BSN4_5_out.Res_0_6, SD_BO_07 := "Sfty_Comm".BSN4_5_out.Res_0_7, SD_BO_08 := "Sfty_Comm".BSN4_5_out.Res_1_0, SD_BO_09 := "Sfty_Comm".BSN4_5_out.Res_1_1, SD_BO_10 := "Sfty_Comm".BSN4_5_out.Res_1_2, SD_BO_11 := "Sfty_Comm".BSN4_5_out.Res_1_3, SD_BO_12 := "Sfty_Comm".BSN4_5_out.Res_1_4, SD_BO_13 := "Sfty_Comm".BSN4_5_out.Res_1_5, SD_BO_14 := "Sfty_Comm".BSN4_5_out.Res_1_6, SD_BO_15 := "Sfty_Comm".BSN4_5_out.Res_1_7, SD_I_00 :=, SD_I_01 :=, SD_DI_00 :=, DINTMODE :=, DP_DP_ID := 116, TIMEOUT := T#1000ms, LADDR := "BSN4_5~01_F-CD_=CRS-=1K1_WAO", ERROR => "Sfty_Status"."CRS_BSN4/5_Fault".Flt, SUBS_ON => "Sfty_Status"."CRS_BSN4/5_Fault".SftyModeDeact, RET_DPRD =>, RET_DPWR =>, DIAG =>)
   END_RUNG
   // the same network as SCL:
   "SENDDP_BSN4_5_DB"(SD_BO_00 := "Sfty_Comm".BSN4_5_out.LiveBit,   // SENDDP
                      SD_BO_01 := "Sfty_Comm".BSN4_5_out.SftyMode,
                      SD_BO_02 := "Sfty_Comm".BSN4_5_out.EmgStop,
                      SD_BO_03 := "Sfty_Comm".BSN4_5_out.InputConvBSN4En,
                      SD_BO_04 := "Sfty_Comm".BSN4_5_out.InputConvBSN5En,
                      SD_BO_05 := "Sfty_Comm".BSN4_5_out.Res_0_5,
                      SD_BO_06 := "Sfty_Comm".BSN4_5_out.Res_0_6,
                      SD_BO_07 := "Sfty_Comm".BSN4_5_out.Res_0_7,
                      SD_BO_08 := "Sfty_Comm".BSN4_5_out.Res_1_0,
                      SD_BO_09 := "Sfty_Comm".BSN4_5_out.Res_1_1,
                      SD_BO_10 := "Sfty_Comm".BSN4_5_out.Res_1_2,
                      SD_BO_11 := "Sfty_Comm".BSN4_5_out.Res_1_3,
                      SD_BO_12 := "Sfty_Comm".BSN4_5_out.Res_1_4,
                      SD_BO_13 := "Sfty_Comm".BSN4_5_out.Res_1_5,
                      SD_BO_14 := "Sfty_Comm".BSN4_5_out.Res_1_6,
                      SD_BO_15 := "Sfty_Comm".BSN4_5_out.Res_1_7,
                      DP_DP_ID := 116,
                      TIMEOUT := T#1000ms,
                      LADDR := "BSN4_5~01_F-CD_=CRS-=1K1_WAO",
                      ERROR => "Sfty_Status"."CRS_BSN4/5_Fault".Flt,
                      SUBS_ON => "Sfty_Status"."CRS_BSN4/5_Fault".SftyModeDeact);
END_REGION

REGION Network 19: *************** Outgoing communication section end ***************
END_REGION
END_FUNCTION_BLOCK
